// Mitsubishi GX Works2 project: 41915063   PLC: Q02/Q02H

PROGRAM MAIN
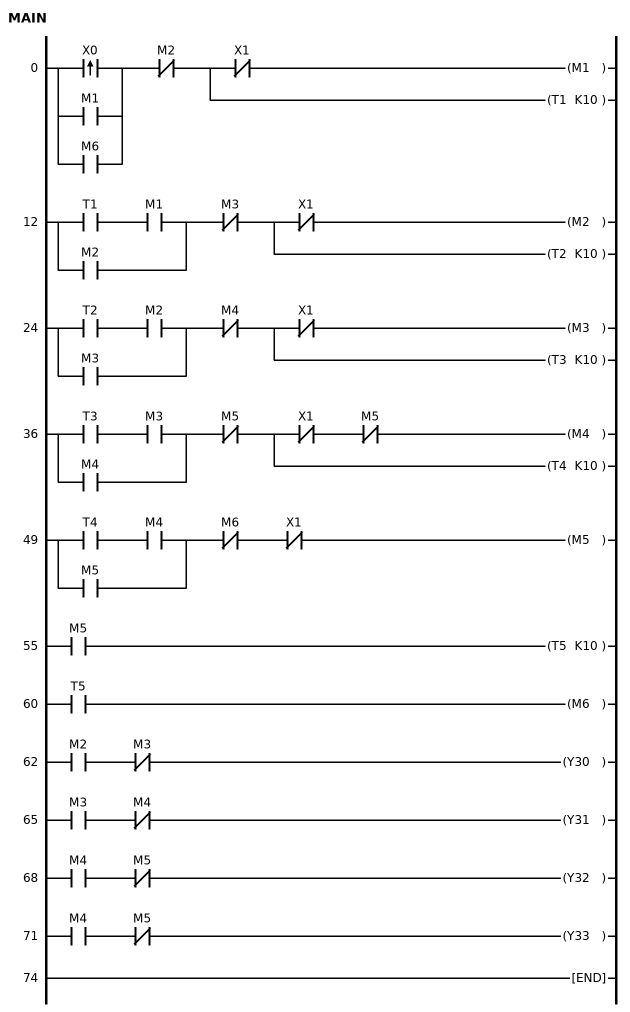
0     LDP     X0
      OR      M1
      OR      M6
      ANI     M2
      MPS
      ANI     X1
      OUT     M1
      MPP
      OUT     T1 K10
12    LD      T1
      AND     M1
      OR      M2
      ANI     M3
      MPS
      ANI     X1
      OUT     M2
      MPP
      OUT     T2 K10
24    LD      T2
      AND     M2
      OR      M3
      ANI     M4
      MPS
      ANI     X1
      OUT     M3
      MPP
      OUT     T3 K10
36    LD      T3
      AND     M3
      OR      M4
      ANI     M5
      MPS
      ANI     X1
      ANI     M5
      OUT     M4
      MPP
      OUT     T4 K10
49    LD      T4
      AND     M4
      OR      M5
      ANI     M6
      ANI     X1
      OUT     M5
55    LD      M5
      OUT     T5 K10
60    LD      T5
      OUT     M6
62    LD      M2
      ANI     M3
      OUT     Y30
65    LD      M3
      ANI     M4
      OUT     Y31
68    LD      M4
      ANI     M5
      OUT     Y32
71    LD      M4
      ANI     M5
      OUT     Y33
74    END
END_PROGRAM
